INTERFACE I_MotionAxisCommonDS402

METHOD DS402StateMachine
VAR_INPUT
END_VAR
END_METHOD

PROPERTY Operational : BOOL
GET
END_GET
SET
END_SET
END_PROPERTY

END_INTERFACE

(* stored: Version 1.1.0.1
   Itf I_MotionAxisCommonDS402: Id {5cfa6b6b-bfba-4af4-97dd-dc8ae67741ad}
   Method DS402StateMachine: Id {f34b87af-faea-4705-b0f9-691a780e3e37}
   Property Operational: Id {58691f2a-6d0a-4bad-9226-70b803c51399}
   Get Get: Id {2bdb4f42-1332-42f1-9883-3120996c5c68}
   Set Set: Id {8db2765c-b1af-4a6b-8530-ac9bd2cb12d3} *)
